PROGRAM TECH_MAIN
VAR
	_app : AppContext;
END_VAR

_app.Run();
_app.RtcSynchronize(TRUE, '', 60);

END_PROGRAM

(* stored: Version 1.1.0.1, ProductVersion 3.1.4024.9
   POU TECH_MAIN: Id {84d391ff-245d-469c-9f07-0280ac5ddd13}, SpecialFunc None *)
